Universal Robots PolyScope program: ur16_control_demo.urp

Program ur16_control_demo (installation=default directory=/home/ur/ursim-current/programs/new folder createdIn=5.11.5.1010327 lastSavedIn=5.11.5.1010327 robotSerialNumber=20195699999)
Calibrated DH parameters: a=[0, -0.4784, -0.36, 0, 0, 0]; d=[0.1807, 0, 0, 0.17415, 0.11985, 0.11655]; alpha=[1.570796, 0, 0, 1.570796, -1.570796, 0]; deltaTheta=[0, 0, 0, 0, 0, 0]
BeforeStart
  connection := False
  Loop While (checkContinuously=false) expression=not connection
    connection := socket_open("172.16.140.1",1201)
Robot Program (runOnlyOnce=false)
  Script: socket_send_string("Anna auto")
  auto := socket_read_string(timeout=0)
  Script: socket_send_string("Anna paketti")
  paketti := socket_read_string(timeout=0)
  Popup Message (haltProgram=false inputType=Variable) variable=paketti
  Wait NoWait
  Script: socket_send_string("paskea")
  Wait Sleep waitTime=2
  Script: socket_send_string("Lastattu")
  Wait NoWait
